{attribute addProperty BoxType "EL3443-0000-0016"}
{attribute addProperty Id "L1_StatusAT %I*L1_Status_EEFC181480100L1_BasicAT %I*L1_Basic_005DC40B6480L1_PowerAT %I*L1_Power_E8C64AA4128160L1_TimingAT %I*L1_Timing_41B415056480L2_StatusAT %I*L2_Status_EEFC181480100L2_BasicAT %I*L2_Basic_005DC40B6480L2_PowerAT %I*L2_Power_E8C64AA4128160L2_TimingAT %I*L2_Timing_41B415056480L3_StatusAT %I*L3_Status_EEFC181480100L3_BasicAT %I*L3_Basic_005DC40B6480L3_PowerAT %I*L3_Power_E8C64AA4128160L3_TimingAT %I*L3_Timing_41B415056480Total_StatusAT %I*Total_Status_F4CDE3E7144180Total_BasicAT %I*Total_Basic_097E4CFE96120Total_ActiveAT %I*Total_Active_7556780A224280Total_L_L_VoltageAT %I*Total_L_L_Voltage_36E7ACB196120WcStateAT %I*WcState_98A4DF7520.250InfoDataAT %I*InfoData_BC63D37F80100"}
{attribute addProperty CRC "3816406624"}
{attribute addProperty SizeInBites "1650"}
{attribute addProperty SizeInBytes "206.25"}
TYPE EL3443_2BD502B5 :
STRUCT
	{attribute addProperty Name "L1_Status"}
	L1_Status : L1_Status_EEFC1814;
	{attribute addProperty Name "L1_Basic"}
	L1_Basic : L1_Basic_005DC40B;
	{attribute addProperty Name "L1_Power"}
	L1_Power : L1_Power_E8C64AA4;
	{attribute addProperty Name "L1_Timing"}
	L1_Timing : L1_Timing_41B41505;
	{attribute addProperty Name "L2_Status"}
	L2_Status : L2_Status_EEFC1814;
	{attribute addProperty Name "L2_Basic"}
	L2_Basic : L2_Basic_005DC40B;
	{attribute addProperty Name "L2_Power"}
	L2_Power : L2_Power_E8C64AA4;
	{attribute addProperty Name "L2_Timing"}
	L2_Timing : L2_Timing_41B41505;
	{attribute addProperty Name "L3_Status"}
	L3_Status : L3_Status_EEFC1814;
	{attribute addProperty Name "L3_Basic"}
	L3_Basic : L3_Basic_005DC40B;
	{attribute addProperty Name "L3_Power"}
	L3_Power : L3_Power_E8C64AA4;
	{attribute addProperty Name "L3_Timing"}
	L3_Timing : L3_Timing_41B41505;
	{attribute addProperty Name "Total_Status"}
	Total_Status : Total_Status_F4CDE3E7;
	{attribute addProperty Name "Total_Basic"}
	Total_Basic : Total_Basic_097E4CFE;
	{attribute addProperty Name "Total_Active"}
	Total_Active : Total_Active_7556780A;
	{attribute addProperty Name "Total_L_L_Voltage"}
	Total_L_L_Voltage : Total_L_L_Voltage_36E7ACB1;
	{attribute addProperty Name "WcState"}
	WcState : WcState_98A4DF75;
	{attribute addProperty Name "InfoData"}
	InfoData : InfoData_BC63D37F;
END_STRUCT
END_TYPE

(* stored: Version 1.2.0.0, ProductVersion 3.1.4024.9
   DUT EL3443_2BD502B5: Id {33af982f-9126-4801-ad73-c49bd1da08ff} *)
